Fanuc KAREL source: wuseturns.kl

PROGRAM wuseturns
%NOLOCKGROUP
VAR
  p : POSITION
  q : POSITION
  i : INTEGER
  r : REAL
BEGIN
  WITH $USE_TURNS = TRUE MOVE TO p
END wuseturns
